// TIA Portal V21 export
// export: Created 2026-08-26T08:43:03.8687053Z, ExportSetting None, DisplayName Totally Integrated Automation Portal, DisplayVersion V21, DisplayName STEP 7 Professional, DisplayVersion V21, DisplayName STEP 7 Safety, DisplayVersion V21, DisplayName Tech WebApplication, DisplayVersion V21, DisplayName WinCC Basic/Comfort/Advanced, DisplayVersion V21
FUNCTION "TASK012A_FC_Callee" : Void   // FC1, LAD
{ S7_Optimized_Access := 'TRUE' }
// stored: SetENOAutomatically false
   VAR_INPUT
      Enable : Bool;
   END_VAR
   VAR_OUTPUT
      Ok : Bool;
   END_VAR
BEGIN

REGION Network 1
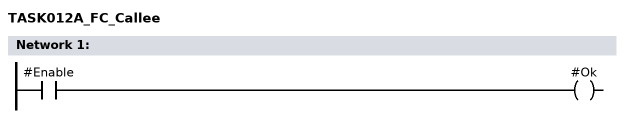
   RUNG wire#powerrail
      Contact( #Enable )
      Coil( #Ok )
   END_RUNG
   // the same network as SCL:
   #Ok := #Enable;
END_REGION
END_FUNCTION
